INTERFACE IPistonGripper

METHOD Close : TcoCore.ITcoTaskStatus
END_METHOD

METHOD Open : TcoCore.ITcoTaskStatus
END_METHOD

END_INTERFACE

(* stored: Version 1.1.0.1, ProductVersion 3.1.4024.6
   Itf IPistonGripper: Id {1dbe9966-81b2-4a54-8a38-b6ae1ee05473}
   Folder Gripper: Id {09630ec4-e465-4e25-9060-0756591cadd2}
   Method Close: Id {5f49f547-446d-461d-8026-5e70873a6dda}
   Method Open: Id {ead70bc3-540c-4017-9dcc-290057385aa6} *)
